PROGRAM prgDataAnaylse
VAR
	windowCheck:FB_Window;
	
END_VAR

//windowCheck	(dataAxis := dataGrab.	,
//			);

END_PROGRAM

(* stored: Version 1.1.0.1, ProductVersion 3.1.4024.11
   POU prgDataAnaylse: Id {5b64e1c3-e236-0a4e-1cd2-9817ef2395fb}, SpecialFunc None *)
